FUNCTION_BLOCK FB_SpindleFunctions IMPLEMENTS I_HMI;

// Spindle VFD control for Invertek Optidrive E3 (240V single phase input, 240V three phase output, 2.2KW) and GMT 400hz 2.2kw 3 HP Spindle using Modbus RTU
VAR_INPUT
    
nSpindleSpeedFromNC     		: UINT;
bManualSpindleOverride  		: BOOL;
bEnable							: BOOL;
bStart							: BOOL;
bReset							: BOOL;
eRequestedState					: E_MachineState;

END_VAR


VAR
	

 eLastState						: E_MachineState;
 bStateEntry					: BOOL;
 
 fbModbusMasterEL           	: ModbusRtuMasterV2_KL6x22B;
 fbSpeedRefScale            	: FB_CTRL_SCALE;
 fbSpeedRefScaleforHMI      	: FB_CTRL_SCALE;
 fbMessage		    			: FB_TcMessage;
 stSpeedRefScaleParams       	: ST_CTRL_SCALE_PARAMS;
 stSpeedRefScaleParamsforHMI	: ST_CTRL_SCALE_PARAMS;
 fScaledSpindleSpeedRef    		: LREAL;
 nModbusReadBlk1    			: ARRAY [1..46] OF INT;
 nModbusReadBlk2    			: ARRAY [129..188] OF INT;
 // Need to put into a modbus DUT
 nModbusID          			: BYTE :=1;
 nModbusReadQty     			: WORD :=24;
 nModbusReadAddr    			: WORD;
 bReadExecute       			: BOOL;
 bDiagExecute       			: BOOL;
 eReadErrorID       			: MODBUS_ERRORS;
 nCbRead            			: UINT;
 bReadBusy          			: BOOL;
 bReadError         			: BOOL;
 bWriteBusy         			: BOOL;
 bWriteError        			: BOOL;
 nCbWrite           			: UINT;
 bResetSerialComm   			: BOOL;
 
 bWriteDriveCommand             : BOOL;
 bWriteDriveSetpoint            : BOOL;
 bWriteAccel_Decel              : BOOL;
 nModbusWriteDriveCommand       : WORD;
 nModbusWriteDriveSetpoint      : INT;
 nModbusWriteDriveAccel_Decel   : UINT;
 trigWriteBusy					: F_TRIG; // When Write Busy goes TRUE to FALSE the Modbus action has completed
 trigReadBusy					: F_TRIG; // When Read Busy goes TRUE to FALSE the Modbus action has completed
 trigReadExecute                : R_TRIG;
 trigWriteExecute               : R_TRIG;
 PulseWriteExecute              : TP;
 
 eVFDErrors         			: E_VFDErrors;
 stSpindleStatus				: ST_SpindleStatus;
 stSpindleParams    			: ST_SpindleParameters;
 stSpindleControl   			: ST_SpindleControl;

// Sequence Enumerations
 nEnableSpindleSeq      		:INT;
 eReadVFDParamsSeq      		:(INIT_FIRST,READ_FIRST_BLOCK,INIT_SECOND,READ_SECOND_BLOCK,FINISH);
 eSetSpindleSpeedSeq    		:(START,SET_ACCEL,SET_SPEED,FINISH_SPEED,START_ENABLE,ENABLE_DRIVE,RESET_DRIVE,FINISH_ENABLE,SPINDLE_ACTIVE);
 eCoastStop             		:(INIT_STOP,ENABLE_STOP,WAIT_FOR_STOPPED,DISABLE_DRIVE,FINISH_STOP);


nManualSpindleSetpoint  		: UINT;
nSpindleSetpoint        		: UINT;

END_VAR

VAR_OUTPUT
    bSpindleAtRequestedSpeed    : BOOL;
	eCurrentState				: E_MachineState;
	bStateDone					: BOOL;
	bReady						: BOOL;
	bBusy						: BOOL;
	bError						: BOOL;
END_VAR

M_ReadParameters();
M_InputMapping();
M_OutputMapping();
M_DriveErrors();
M_HMI_In();
M_HMI_Out();
StateFollower();

METHOD M_ActiveSpeedChange : BOOL
VAR_INPUT
END_VAR
IF stSpindleStatus.nSpeedRefSetpoint <> nModbusWriteDriveSetpoint THEN
    fbModbusMasterEL.WriteSingleRegister(   
                                                  UnitID:=1,
                                                  Quantity:=1,
                                                  MBAddr:=1,
                                                  cbLength:=SIZEOF(nModbusWriteDriveSetpoint),
                                                  pMemoryAddr:=ADR(nModbusWriteDriveSetpoint),
                                                  Execute:=TRUE,
                                                  Timeout:=T#400MS,
                                                  Busy => bWriteBusy );      
END_IF
END_METHOD

METHOD M_CoastStop : BOOL
VAR_INPUT
    bExecute    : BOOL;
END_VAR
CASE eCoastStop OF


 INIT_STOP:

    M_CoastStop := FALSE;
    stSpindleControl.bCoastStopRequest  := FALSE;
    IF NOT stSpindleControl.bCoastStopRequest AND bExecute THEN
        PulseWriteExecute(IN:=FALSE);
        eCoastStop:=ENABLE_STOP;
	END_IF 
    
ENABLE_STOP:

    stSpindleControl.bCoastStopRequest := TRUE;
    stSpindleControl.bRunEnable := FALSE;
    //trigWriteExecute(CLK:=stSpindleControl.bCoastStopRequest);
    PulseWriteExecute(IN:=stSpindleControl.bCoastStopRequest,PT:=T#250MS);
    fbModbusMasterEL.WriteSingleRegister(   
                                          UnitID:=1,
                                          Quantity:=1,
                                          MBAddr:=0,
                                          cbLength:=SIZEOF(nModbusWriteDriveCommand),
                                          pMemoryAddr:=ADR(nModbusWriteDriveCommand),
                                          Execute:=PulseWriteExecute.Q,
                                          Timeout:=T#300MS,
										  Busy => bWriteBusy );
	 trigWriteBusy(CLK := bWriteBusy); 
     IF trigWriteBusy.Q THEN
        	eCoastStop:=WAIT_FOR_STOPPED;
        	stSpindleControl.bCoastStopRequest := FALSE;
     END_IF
     
WAIT_FOR_STOPPED:
    IF stSpindleStatus.nOutputFreq <= 0.1 THEN
        PulseWriteExecute(IN:=FALSE);
        eCoastStop:=DISABLE_DRIVE; 
     END_IF
    
 
DISABLE_DRIVE:

    stSpindleControl.bRunEnable := FALSE;
    stSpindleControl.bCoastStopRequest := FALSE; 
    trigWriteExecute(CLK:=NOT stSpindleControl.bRunEnable);
    PulseWriteExecute(IN:=TRUE,PT:=T#100MS);
    fbModbusMasterEL.WriteSingleRegister(   
                                          UnitID:=1,
                                          Quantity:=1,
                                          MBAddr:=0,
                                          cbLength:=SIZEOF(nModbusWriteDriveCommand),
                                          pMemoryAddr:=ADR(nModbusWriteDriveCommand),
                                          Execute:= PulseWriteExecute.Q,
                                          Timeout:=T#300MS,
										  Busy => bWriteBusy);
	 trigWriteBusy(CLK := bWriteBusy); 
     IF trigWriteBusy.Q THEN
        PulseWriteExecute(IN:=FALSE);
     	eCoastStop:=FINISH_STOP;  
     END_IF 

FINISH_STOP:
	IF NOT stSpindleControl.bRunEnable THEN
    	stSpindleControl.bCoastStopRequest := FALSE;
    	fbMessage.CreateEx(TC_Events.CNC_Events.Spindle_Stopped,0); 
    	fbMessage.Send(0);
    	eCoastStop :=INIT_STOP;
    	M_CoastStop:=TRUE;
    	bExecute := FALSE;
	END_IF
   
END_CASE;
END_METHOD

METHOD M_DriveErrors : BOOL
VAR_INPUT
END_VAR
eVFDErrors:= stSpindleStatus.nErrorCode;
END_METHOD

METHOD M_Enable : BOOL
VAR_INPUT
    bExecute    : BOOL;
END_VAR
CASE nEnableSpindleSeq OF
    
0:
    M_Enable:=FALSE;
    stSpindleControl.bRunEnable := FALSE;
    stSpindleControl.bResetReq  := FALSE;
    IF NOT stSpindleControl.bRunEnable AND NOT stSpindleControl.bResetReq AND bExecute THEN
        nEnableSpindleSeq:=5;
	END_IF 
    
5:

    stSpindleControl.bRunEnable := TRUE;

    fbModbusMasterEL.WriteSingleRegister(   
                                                                UnitID:=1,
                                                                Quantity:=1,
                                                                MBAddr:=1,
                                                                cbLength:=SIZEOF(nModbusWriteDriveCommand),
                                                                pMemoryAddr:=ADR(nModbusWriteDriveCommand),
                                                                Execute:=TRUE,
                                                                Timeout:=T#400MS, ); 
     IF stSpindleStatus.bDriveEnabled AND stSpindleStatus.bDriveReady THEN 
        nEnableSpindleSeq:=20;
     ELSE
        nEnableSpindleSeq:=10;   
     END_IF 
                                                    
10:
    
    stSpindleControl.bRunEnable:= TRUE;
    stSpindleControl.bResetReq := TRUE;

    fbModbusMasterEL.WriteSingleRegister(   
                                                                UnitID:=1,
                                                                Quantity:=1,
                                                                MBAddr:=1,
                                                                cbLength:=SIZEOF(nModbusWriteDriveCommand),
                                                                pMemoryAddr:=ADR(nModbusWriteDriveCommand),
                                                                Execute:=TRUE,
                                                                Timeout:=T#400MS, );
     IF stSpindleStatus.bDriveEnabled AND stSpindleStatus.bDriveReady THEN 
          nEnableSpindleSeq:=FINISH_ENABLE;
     END_IF 

20:

   // stSpindleControl.bRunEnable := FALSE;
    stSpindleControl.bResetReq  := FALSE;
    fbMessage.CreateEx(TC_Events.CNC_Events.Spindle_Active,0); 
    fbMessage.Send(0);
    nEnableSpindleSeq :=0;
    M_Enable:=TRUE;
    bExecute := FALSE;

END_CASE
END_METHOD

METHOD M_FastStop : BOOL
VAR_INPUT
    bExecute    : BOOL;
END_VAR
END_METHOD

METHOD M_HMI_In : BOOL
// Trigger a state machine reset in the Read Parameters block to reset spindle comms
bResetSerialComm:= stHMI_In.bResetSerialComm;
bManualSpindleOverride := stHMI_In.bManualSpindleOverride;
nManualSpindleSetpoint := stHMI_In.nManualSpindleSetpoint;

(*IF stHMI_In.bSpindleSpeedExecute AND stHMI_In.bManualSpindleOverride THEN     
     bSpindleSetManually := M_SetSpeed();
     IF bSpindleSetManually THEN
         stHMI_In.bSpindleSpeedExecute:=FALSE;
	 END_IF
END_IF*)
END_METHOD


METHOD M_HMI_Out : BOOL
// Map VFD status information to HMI struct
stHMI_Out.nSpeedRefSetpoint	    := stSpindleStatus.nSpeedRefSetpoint;	  
stHMI_Out.nRampControlTime      := stSpindleStatus.nRampControlTime;    
stHMI_Out.sErrorCode		    := TO_STRING(eVFDErrors);	 
stHMI_Out.bDriveRunning         := stSpindleStatus.bDriveRunning; 
stHMI_Out.bDriveFault           := stSpindleStatus.bDriveFault;   
stHMI_Out.bStandbyMode          := stSpindleStatus.bStandbyMode;  
stHMI_Out.bDriveReady           := stSpindleStatus.bDriveReady;   
stHMI_Out.nOutputFreq		    := stSpindleStatus.nOutputFreq;	 
stHMI_Out.nMotorCurrent		    := stSpindleStatus.nMotorCurrent;
stHMI_Out.nMotorTorque          := stSpindleStatus.nMotorTorque; 
stHMI_Out.nMotorPower           := stSpindleStatus.nMotorPower;  
stHMI_Out.bDigitalInput1  	    := stSpindleStatus.nDigitalInputSts.0;
stHMI_Out.bDigitalInput2  	    := stSpindleStatus.nDigitalInputSts.1;
stHMI_Out.bDigitalInput3  	    := stSpindleStatus.nDigitalInputSts.2;    
stHMI_Out.bDigitalInput4  	    := stSpindleStatus.nDigitalInputSts.3;
stHMI_Out.bDriveEnabled         := stSpindleStatus.bDriveEnabled;       
stHMI_Out.nDCBusVoltage		    := stSpindleStatus.nDCBusVoltage;		     
stHMI_Out.nDrivePowerStageTemp  := stSpindleStatus.nDrivePowerStageTemp;
stHMI_Out.bRelayOutputStatus    := stSpindleStatus.nRelayOutputStatus.0;   
stHMI_Out.nKWHourMeter          := stSpindleStatus.nKWHourMeter;  
stHMI_Out.nRuntimeHours         := stSpindleStatus.nRuntimeHours;
stHMI_Out.nRuntimeMinutes       := stSpindleStatus.nRuntimeMinutes;
stHMI_Out.nInternalDriveTemp    := stSpindleStatus.nInternalDriveTemp;  
stHMI_Out.nOutputVoltage        := stSpindleStatus.nOutputVoltage;
// Map VFD Parameter information to HMI struct
stHMI_Out.nMaxSpeedLimit		:= stSpindleParams.nMaxSpeedLimit;
stHMI_Out.nMinSpeedLimit	    := stSpindleParams.nMinSpeedLimit;
stHMI_Out.fAccelRampTime		:= UINT_TO_REAL(stSpindleParams.nAccelRampTime)/100;
stHMI_Out.nDecelRampTime		:= stSpindleParams.nDecelRampTime;
stHMI_Out.nStopMode			    := stSpindleParams.nStopMode;
stHMI_Out.nMotorRatedVoltage	:= stSpindleParams.nMotorRatedVoltage;
stHMI_Out.nMotorRatedCurrent    := stSpindleParams.nMotorRatedCurrent;
stHMI_Out.nMotorRatedFrequency  := stSpindleParams.nMotorRatedFrequency;
stHMI_Out.nMotorRatedSpeed      := stSpindleParams.nMotorRatedSpeed;
stHMI_Out.nApplicationMode      := stSpindleParams.nApplicationMode;
stHMI_Out.nRelayOutputFunction  := stSpindleParams.nRelayOutputFunction;
stHMI_Out.nUserPGain            := stSpindleParams.nUserPGain;
stHMI_Out.nUserIConstant        := stSpindleParams.nUserIConstant;
stHMI_Out.nMotorControlMode     := stSpindleParams.nMotorControlMode;
stHMI_Out.nMaximumCurrentLimit  := stSpindleParams.nMaximumCurrentLimit;

//// Map Modbus Comms information to HMI struct

stHMI_Out.sReadErrorID := TO_STRING(eReadErrorID);
stHMI_Out.bSpindleAtRequestedSpeed := bSpindleAtRequestedSpeed;

stSpeedRefScaleParamsforHMI.fInMax:= 4000.0 ;
stSpeedRefScaleParamsforHMI.fInMin:=  1333.0;
stSpeedRefScaleParamsforHMI.fOutMax:=  24000.0;
stSpeedRefScaleParamsforHMI.fOutMin:=  8000.0;
stSpeedRefScaleParamsforHMI.tCtrlCycleTime:= T#2MS  ;
stSpeedRefScaleParamsforHMI.tTaskCycleTime:=  T#2MS ;

// Scale Spindle Speed Setpoint From RPM to Hz


fbSpeedRefScaleforHMI(
                fIn:=stSpindleStatus.nSpeedRefSetpoint,
                fOut=>stHMI_Out.fScaledSpindleSpeedRef,
                eErrorId=>,
                bError=>,
                stParams:=stSpeedRefScaleParamsforHMI,
                                                    );
END_METHOD

METHOD M_InitalizeParameters : BOOL
VAR_INPUT
END_VAR
END_METHOD

METHOD M_InputMapping : BOOL
VAR_INPUT
END_VAR
// Map Spindle Status
stSpindleStatus.nControlWord        := INT_TO_WORD(nModbusReadBlk1[1]);	   
stSpindleStatus.nSpeedRefSetpoint	:= nModbusReadBlk1[2];
stSpindleStatus.nRampControlTime    := INT_TO_UINT(nModbusReadBlk1[4]);
stSpindleStatus.bDriveRunning       := nModbusReadBlk1[6].0;
stSpindleStatus.bDriveFault         := nModbusReadBlk1[6].1;
stSpindleStatus.bStandbyMode        := nModbusReadBlk1[6].5;
stSpindleStatus.bDriveReady         := nModbusReadBlk1[6].6;                                  
stSpindleStatus.nErrorCode			:= INT_TO_BYTE(SHR(nModbusReadBlk1[6],8)); 
stSpindleStatus.nOutputFreq			:= nModbusReadBlk1[7];	
stSpindleStatus.nMotorCurrent		:= INT_TO_UINT(nModbusReadBlk1[8]);  
stSpindleStatus.nMotorTorque        := nModbusReadBlk1[9];  
stSpindleStatus.nMotorPower         := INT_TO_UINT(nModbusReadBlk1[10]);  
stSpindleStatus.nDigitalInputSts	:= INT_TO_WORD(nModbusReadBlk1[11]);
stSpindleStatus.bDriveEnabled       := nModbusReadBlk1[11].0;	
stSpindleStatus.nDCBusVoltage		:= INT_TO_UINT(nModbusReadBlk1[23]); 
stSpindleStatus.nDrivePowerStageTemp:= nModbusReadBlk1[24];	
stSpindleStatus.nRelayOutputStatus  := INT_TO_WORD(nModbusReadBlk1[29]);  
stSpindleStatus.nKWHourMeter        := INT_TO_UINT(nModbusReadBlk1[32]);  
stSpindleStatus.nRuntimeHours       := INT_TO_UINT(nModbusReadBlk1[34]);  
stSpindleStatus.nRuntimeMinutes     := INT_TO_UINT(nModbusReadBlk1[35]);
stSpindleStatus.nInternalDriveTemp  := nModbusReadBlk1[39];
stSpindleStatus.nOutputVoltage      := INT_TO_UINT(nModbusReadBlk1[43]);

// Map Spindle Parameters

stSpindleParams.nMaxSpeedLimit		:= INT_TO_UINT(nModbusReadBlk2[129]);
stSpindleParams.nMinSpeedLimit	    := INT_TO_UINT(nModbusReadBlk2[130]);
stSpindleParams.nAccelRampTime		:= INT_TO_UINT(nModbusReadBlk2[131]);
stSpindleParams.nDecelRampTime		:= INT_TO_UINT(nModbusReadBlk2[132]);
stSpindleParams.nStopMode			:= INT_TO_UINT(nModbusReadBlk2[133]);
stSpindleParams.nMotorRatedVoltage	:= INT_TO_UINT(nModbusReadBlk2[135]);
stSpindleParams.nMotorRatedCurrent  := INT_TO_UINT(nModbusReadBlk2[136]);
stSpindleParams.nMotorRatedFrequency:= INT_TO_UINT(nModbusReadBlk2[137]);
stSpindleParams.nMotorRatedSpeed    := INT_TO_UINT(nModbusReadBlk2[138]);
stSpindleParams.nApplicationMode    := INT_TO_UINT(nModbusReadBlk2[141]);
stSpindleParams.nRelayOutputFunction:= INT_TO_UINT(nModbusReadBlk2[146]);
stSpindleParams.nUserPGain          := INT_TO_UINT(nModbusReadBlk2[169]);
stSpindleParams.nUserIConstant      := INT_TO_UINT(nModbusReadBlk2[170]);
stSpindleParams.nMotorControlMode   := INT_TO_UINT(nModbusReadBlk2[179]);
stSpindleParams.nMaximumCurrentLimit:= INT_TO_UINT(nModbusReadBlk2[182]);

IF bManualSpindleOverride THEN  
    nSpindleSetpoint    := nManualSpindleSetpoint;   
ELSE
    nSpindleSetpoint    := nSpindleSpeedFromNC;
END_IF
END_METHOD

METHOD M_OutputMapping : BOOL
VAR_INPUT
END_VAR
// Map Spindle Control

stSpeedRefScaleParams.fInMax:= 24000.0 ;
stSpeedRefScaleParams.fInMin:=  8000.0;
stSpeedRefScaleParams.fOutMax:=  4000.0;
stSpeedRefScaleParams.fOutMin:=  1333.0;
stSpeedRefScaleParams.tCtrlCycleTime:= T#2MS  ;
stSpeedRefScaleParams.tTaskCycleTime:=  T#2MS ;

// Scale Spindle Speed Setpoint From RPM to Hz
fbSpeedRefScale(
                fIn:=nSpindleSetpoint,
                fOut=>fScaledSpindleSpeedRef,
                eErrorId=>,
                bError=>,
                stParams:=stSpeedRefScaleParams,
                                                    );                                                                                                 
                                                    
nModbusWriteDriveCommand.0 :=stSpindleControl.bRunEnable;
nModbusWriteDriveCommand.1 :=stSpindleControl.bFastStopReq;
nModbusWriteDriveCommand.2 :=stSpindleControl.bResetReq;
nModbusWriteDriveCommand.3 :=stSpindleControl.bCoastStopRequest;

nModbusWriteDriveSetpoint  :=LREAL_TO_INT(fScaledSpindleSpeedRef);

nModbusWriteDriveAccel_Decel :=stSpindleControl.nRampControlTime;
END_METHOD

METHOD M_ReadParameters : BOOL
VAR_INPUT
END_VAR
IF bResetSerialComm THEN
    eReadVFDParamsSeq := FINISH;    
END_IF
    CASE eReadVFDParamsSeq OF
        
        INIT_FIRST:
            fbModbusMasterEL.ReadRegs(Execute:=bReadExecute);
            eReadVFDParamsSeq:=READ_FIRST_BLOCK;
            bReadExecute:=FALSE;
            trigReadExecute(CLK:=bReadExecute);
        
        READ_FIRST_BLOCK:
        IF NOT GVL.stHMI_Out.bBufferFull THEN
        bReadExecute:=TRUE;
        trigReadExecute(CLK:=bReadExecute);
        END_IF
            fbModbusMasterEL.ReadRegs(
                                    UnitID:= 1, 
                                    Quantity:= 45, 
                                    MBAddr:= 0, 
                                    cbLength:= SIZEOF(nModbusReadBlk1), 
                                    pMemoryAddr:= ADR(nModbusReadBlk1), 
                                    Execute:= trigReadExecute.Q AND NOT PulseWriteExecute.Q, 
                                    Timeout:= T#300MS, 
                                    Busy=> bReadBusy, 
                                    Error=> bReadError, 
                                    ErrorId=> eReadErrorID, 
                                    cbRead=> nCbRead);
									
			 trigReadBusy(CLK:=bReadBusy);						
             IF trigReadBusy.Q AND NOT bReadError THEN
             	bReadExecute:=FALSE;                       
             	eReadVFDParamsSeq:=INIT_SECOND;
             END_IF 
             
        INIT_SECOND:
		
           fbModbusMasterEL.ReadRegs(Execute:=bReadExecute);
           eReadVFDParamsSeq:=READ_SECOND_BLOCK;
           bReadExecute:=FALSE;
           trigReadExecute(CLK:=bReadExecute); 
    
        READ_SECOND_BLOCK:
            IF NOT GVL.stHMI_Out.bBufferFull THEN
            bReadExecute:=TRUE;
            trigReadExecute(CLK:=bReadExecute);
            END_IF
            fbModbusMasterEL.ReadRegs(
                                    UnitID:= 1, 
                                    Quantity:= 59, 
                                    MBAddr:= 128, 
                                    cbLength:= SIZEOF(nModbusReadBlk2), 
                                    pMemoryAddr:= ADR(nModbusReadBlk2), 
                                    Execute:= trigReadExecute.Q AND NOT PulseWriteExecute.Q, 
                                    Timeout:= T#300MS, 
                                    Busy=> bReadBusy, 
                                    Error=> bReadError, 
                                    ErrorId=> eReadErrorID, 
                                    cbRead=> nCbRead);
                                    
             trigReadBusy(CLK:=bReadBusy);						
             IF trigReadBusy.Q AND NOT bReadError THEN                       
             	eReadVFDParamsSeq:=FINISH;
             END_IF 
        
        FINISH:
        bReadExecute:=FALSE;
        trigReadExecute(CLK:=bReadExecute);    
        eReadVFDParamsSeq:=INIT_FIRST;
    
    END_CASE
END_METHOD

METHOD M_ResetDriveError : BOOL
VAR_INPUT
END_VAR
(*                                                    
RESET_DRIVE:
    bWriteTimerExec := TRUE;
    stSpindleControl.bRunEnable:= TRUE;
    stSpindleControl.bResetReq := TRUE;

    fbModbusMasterEL.WriteSingleRegister(   
                                                                UnitID:=1,
                                                                Quantity:=1,
                                                                MBAddr:=0,
                                                                cbLength:=SIZEOF(nModbusWriteDriveCommand),
                                                                pMemoryAddr:=ADR(nModbusWriteDriveCommand),
                                                                Execute:=TRUE,
                                                                Timeout:=T#400MS, );
     IF stSpindleControl.bRunEnable AND stSpindleControl.bResetReq AND tWriteTimer.Q THEN 
          eSetSpindleSpeedSeq:=FINISH_ENABLE;
     END_IF 
*)
END_METHOD

METHOD M_SetSpeed : BOOL
VAR_INPUT
    bExecute    : BOOL;
END_VAR
 
CASE eSetSpindleSpeedSeq OF
    
START:
    M_SetSpeed:=FALSE;
    bWriteDriveSetpoint := FALSE;
    bWriteAccel_Decel := FALSE;
    IF stSpindleStatus.bDriveReady AND stSpindleStatus.bDriveEnabled AND bExecute THEN
        eSetSpindleSpeedSeq:=SET_ACCEL;
        trigWriteExecute(CLK:=FALSE);
        PulseWriteExecute(IN:=FALSE);
	END_IF
    
SET_ACCEL:
    bWriteAccel_Decel:=TRUE;
    //trigWriteExecute(CLK:=bWriteAccel_Decel);
    PulseWriteExecute(IN:=bWriteAccel_Decel,PT:=T#300MS);
    fbModbusMasterEL.WriteSingleRegister(   
                                          UnitID:=1,
                                          Quantity:=1,
                                          MBAddr:=3,
                                          cbLength:=SIZEOF(nModbusWriteDriveAccel_Decel),
                                          pMemoryAddr:=ADR(nModbusWriteDriveAccel_Decel),
                                          Execute:=PulseWriteExecute.Q,
                                          Timeout:=T#300MS,
                                          Busy => bWriteBusy);      
	trigWriteBusy(CLK := bWriteBusy); 
    IF trigWriteBusy.Q THEN
		bWriteAccel_Decel := FALSE;
        eSetSpindleSpeedSeq:=SET_SPEED;
        //trigWriteExecute(CLK:=FALSE);
        PulseWriteExecute(IN:=FALSE);
    END_IF
                                                    
SET_SPEED:
    bWriteDriveSetpoint:=TRUE;
    //trigWriteExecute(CLK:=bWriteDriveSetpoint);
    PulseWriteExecute(IN:=bWriteDriveSetpoint,PT:=T#300MS);
    fbModbusMasterEL.WriteSingleRegister(   
                                                  UnitID:=1,
                                                  Quantity:=1,
                                                  MBAddr:=1,
                                                  cbLength:=SIZEOF(nModbusWriteDriveSetpoint),
                                                  pMemoryAddr:=ADR(nModbusWriteDriveSetpoint),
                                                  Execute:=PulseWriteExecute.Q,
                                                  Timeout:=T#300MS,
                                                  Busy => bWriteBusy);      
	trigWriteBusy(CLK := bWriteBusy); 
    IF trigWriteBusy.Q THEN
		bWriteDriveSetpoint := FALSE;
        trigWriteExecute(CLK:=FALSE);
        eSetSpindleSpeedSeq:=FINISH_SPEED;
    END_IF

FINISH_SPEED:
          fbMessage.CreateEx(TC_Events.CNC_Events.Spindle_Speed_Updated,0); 
          fbMessage.Send(0);
          bWriteDriveSetpoint := FALSE;
          bWriteAccel_Decel := FALSE; 
          eSetSpindleSpeedSeq:=START_ENABLE;

START_ENABLE:

    stSpindleControl.bRunEnable := FALSE;
    stSpindleControl.bResetReq  := FALSE;
    IF NOT stSpindleControl.bRunEnable AND NOT stSpindleControl.bResetReq THEN
        eSetSpindleSpeedSeq:=ENABLE_DRIVE;
        //trigWriteExecute(CLK := FALSE);
        PulseWriteExecute(IN:=FALSE);
	END_IF 
    
ENABLE_DRIVE:

    stSpindleControl.bRunEnable := TRUE;
    //trigWriteExecute(CLK:=stSpindleControl.bRunEnable);
    PulseWriteExecute(IN:=stSpindleControl.bRunEnable,PT:=T#300MS);
    fbModbusMasterEL.WriteSingleRegister(   
                                          UnitID:=1,
                                          Quantity:=1,
                                          MBAddr:=0,
                                          cbLength:=SIZEOF(nModbusWriteDriveCommand),
                                          pMemoryAddr:=ADR(nModbusWriteDriveCommand),
                                          Execute:=PulseWriteExecute.Q,
                                          Timeout:=T#300MS,
										  Busy => bWriteBusy);
	 trigWriteBusy(CLK := bWriteBusy); 
     IF trigWriteBusy.Q AND stSpindleControl.bRunEnable THEN
		//stSpindleControl.bRunEnable := FALSE; 
        trigWriteExecute(CLK := FALSE);
        eSetSpindleSpeedSeq:=FINISH_ENABLE; 
     END_IF 

FINISH_ENABLE:
 
	IF stSpindleStatus.bDriveRunning AND stSpindleStatus.nSpeedRefSetpoint = nModbusWriteDriveSetpoint THEN
    	M_SetSpeed:=TRUE;
		eSetSpindleSpeedSeq :=START;
		fbMessage.CreateEx(TC_Events.CNC_Events.Spindle_Active,0); 
    	fbMessage.Send(0);
	END_IF
END_CASE
END_METHOD

METHOD StateFollower : BOOL
VAR_INPUT
END_VAR
bStateEntry := (eCurrentState <> eLastState);

CASE eCurrentState OF

    E_MachineState.IDLE:
        // Follower Logic: If Master requests STARTING or EXECUTE, we move.
        IF eRequestedState = E_MachineState.STARTING OR eRequestedState = E_MachineState.EXECUTE THEN
            eCurrentState := E_MachineState.STARTING;
        END_IF
        
    E_MachineState.STARTING:
        // We stay here until the Method confirms we are up to speed
        IF M_SetSpeed(bExecute := bStateEntry) THEN
            eCurrentState := E_MachineState.EXECUTE;
			bStateDone := TRUE;
        END_IF
        
    E_MachineState.EXECUTE:
        // Global Check: If VFD trips, jump to Aborting
        IF eVFDErrors <> 0 THEN
            eCurrentState := E_MachineState.ABORTING;
        
        // Follower Logic: If Master moves to COMPLETING or STOPPING, we follow
        ELSIF eRequestedState = E_MachineState.COMPLETING OR eRequestedState = E_MachineState.STOPPED THEN
            eCurrentState := E_MachineState.COMPLETING; // Use your ramp-down logic
			bStateDone := TRUE;
        END_IF
    
    E_MachineState.COMPLETING:
        // Action: Coast/Ramp down
        IF M_CoastStop(bExecute := bStateEntry) THEN
             eCurrentState := E_MachineState.IDLE;
			 bStateDone := TRUE;
        END_IF

    E_MachineState.ABORTING:
        // Force an immediate stop
        IF M_FastStop(bExecute := bStateEntry) THEN
            eCurrentState := E_MachineState.ABORTED;
			bStateDone := TRUE;
        END_IF

    E_MachineState.ABORTED:
        // Follower Logic: Only exit if the Master requests RESETTING
        IF eRequestedState = E_MachineState.RESETTING AND (eVFDErrors = 0) THEN
            eCurrentState := E_MachineState.IDLE;
			bStateDone := TRUE;
            // Clear message logic here...
        END_IF

END_CASE

eLastState := eCurrentState; // Don't forget to update this at the end!
// Reset bStateDone if the Master changes the request
IF eCurrentState <> eRequestedState THEN
    bStateDone := FALSE;
END_IF
END_METHOD

END_FUNCTION_BLOCK

(* stored: Version 1.1.0.1
   POU FB_SpindleFunctions: Id {d33eb993-f1a5-484e-9d4d-ae7861108719}, SpecialFunc None
   Folder State Machine: Id {3873f6fc-5a3d-4287-91cc-401f0647d882}
   Method M_ActiveSpeedChange: Id {8c91d8ac-e153-43a1-8a22-2e9bee5bdf48}
   Method M_CoastStop: Id {f02bd68b-a8e2-4168-ba64-5310fb0ed017}
   Method M_DriveErrors: Id {5214dc49-55b0-4763-8ae7-946b59ed4930}
   Method M_Enable: Id {00000b6e-cbd2-4a72-a802-b97127827ff0}
   Method M_FastStop: Id {de81cf2d-b911-460a-8df3-f1e95bcc53de}
   Method M_HMI_In: Id {7023150e-5dba-40bd-b6bf-f2224d2f965b}
   Method M_HMI_Out: Id {7a175b83-8eaa-4aad-b855-25562de10eb8}
   Method M_InitalizeParameters: Id {02772613-62d0-43d8-a964-5b84e2c9be3d}
   Method M_InputMapping: Id {83d865f8-d7ae-49d7-a6f4-fcb7ec40a615}
   Method M_OutputMapping: Id {9f934105-dd30-493a-85e5-9cee50265608}
   Method M_ReadParameters: Id {a233cd63-eba1-4191-8645-5e9df383ad75}
   Method M_ResetDriveError: Id {6a769b7b-415c-4e9d-90e8-e0d6e861e949}
   Method M_SetSpeed: Id {0d91e475-0382-4cfa-b413-5ce8843a481a}
   Method StateFollower: Id {41ddc753-3b32-4bf2-8aa9-5484efb3ad6b} *)
